{attribute 'qualified_only'}
{attribute 'strict'}
TYPE E_TransportTube :
(
	BO4 := 0, // Output tube 1
	BI1 := 1 // Input tube 1
);
END_TYPE

(* stored: Version 1.1.0.1, ProductVersion 3.1.4024.0
   DUT E_TransportTube: Id {bcb0bf0b-15c7-0883-24e2-59f0f27b9ba3} *)
